PROGRAM P_Demo_FB_SoEAX5000ParkAxis
VAR
    fbAX5000ParkAxis   : FB_SoEAX5000ParkAxis; // AX5000 驻留/释放 FB 实例
    axisOptionStation  : AXIS_REF; // AX5000 可选工位轴引用；未装电机的通道
    rtParkTrig         : R_TRIG; // 把电平转上升沿
    bParkReq           : BOOL := FALSE; // 在线写 TRUE 触发一次驻留/释放
    eRequestedParkMode : E_ParkMode; // 在线选 eParkMode_Park / eParkMode_Release
    bParkBusy          : BOOL;
    bParkError         : BOOL;
    nParkErrorID       : UDINT;
END_VAR

// =============================================================================
// 场景：AX5000 驱动的模块化机器某可选工位本批次没装电机。开机时把该通道
//       驻留掉，避免它因缺反馈报错导致整机起不来；装上电机后再释放。
//
// 价值：1) 缺电机的 AX5000 通道驻留后不报反馈错误，机器在缺配置下能启动
//       2) AX5000 专用接口直达（也可用硬件无关的 FB_ParkAxis）
//       3) 运行期动态驻留/释放，免为每种配置维护单独 NC 工程
//
// !! 安全：对多通道 AX5000，驻留/激活某通道前必须先关闭该设备所有通道的
//          控制器使能，否则其它通道的轴会被意外停掉。
//
// 验证步骤：
//   1. System Manager 配好 AX5000 NC 轴并 Link 给 axisOptionStation，引用 Tc2_MC2_Drive
//   2. 确认 AX5000 固件 ≥ v2.12 b0001 且库 ≥ V3.3.21.0
//   3. 对该设备所有通道先 MC_Power(Enable := FALSE) 关使能
//   4. Add Existing Item (.TcPOU) 选本文件，加进 PlcTask，编译登录
//   5. 在线把 eRequestedParkMode 设为 eParkMode_Park，写 bParkReq := TRUE
//   6. 等 bParkBusy 落回 FALSE 且 bParkError = FALSE 即驻留成功
//   7. 装上电机后把 eRequestedParkMode 改为 eParkMode_Release 再触发一次
//   8. 若 bParkError = TRUE，看 nParkErrorID 对照 ADS Return Codes 表
// =============================================================================

// 用 R_TRIG 把"持续按住的 TRUE"转成真正的上升沿
rtParkTrig(CLK := bParkReq);

// 单次调用：Mode 来自在线选择；Axis 是 VAR_IN_OUT 必传
// 本 FB 无 Done，靠 Busy 落回 FALSE 且 Error=FALSE 判成功
fbAX5000ParkAxis(
    Execute := rtParkTrig.Q,
    Mode    := eRequestedParkMode,
    Axis    := axisOptionStation,
    Busy    => bParkBusy,
    Error   => bParkError,
    ErrorID => nParkErrorID
);

END_PROGRAM

(* stored: Version 1.1.0.1, ProductVersion 3.1.4024.5
   POU P_Demo_FB_SoEAX5000ParkAxis: Id {bab6232c-9623-51b1-9e4d-0e6bf61c67df}, SpecialFunc None *)
